// TwinCAT 3 PLC project Untitled1
// ProgramVersion: 3.1.4026.17
// libraries:
//   Tc2_Standard, * (Beckhoff Automation GmbH)
//   Tc2_System, * (Beckhoff Automation GmbH)
// project tree:
//   DUTs/ E_CompressionStages.TcDUT, E_InletToSystem.TcDUT, E_OutletNumber.TcDUT, E_TankBundleNumber.TcDUT, E_ErrorState.TcDUT, E_SolenoidState.TcDUT, ST_AnalogPressureTemp.TcDUT, ST_Path.TcDUT, ST_SolenoidConfig.TcDUT
//   GVLs/ GVL_HMI.TcGVL, GVL_IO.TcGVL
//   / PlcTask.TcTTO
//   POUs/ FB_Device.TcPOU, FB_Matrix.TcPOU, FB_PressureTransducer.TcPOU, FB_Solenoid.TcPOU, MAIN.TcPOU
// real-time tasks:
//   TASK PlcTask: cycle T#10ms, priority 20, ADS port 350
// I/O:
//   DEVICE Node 05 (disabled), AmsNetId 192.168.1.166.2.1
//     Node 05S0 [EK1100 EtherCAT Coupler (2A E-Bus)]
//       Node 05S2 [EL3058 8Ch. Ana. Input 4-20mA]
//       Node 05S4 [EL3058 8Ch. Ana. Input 4-20mA]
//       Node 05S6 [EL3058 8Ch. Ana. Input 4-20mA]
//       Node 05S8 [EL3058 8Ch. Ana. Input 4-20mA]
//       Node 05S10 [EL3058 8Ch. Ana. Input 4-20mA]
//       Node 05S11 [EL1904, 4 Ch. Safety Input 24V, TwinSAFE]
//         modules: Module 1 (FSOES)
//   DEVICE Node 06 (disabled), AmsNetId 192.168.1.166.3.1
//     Node 06S0 [EK1100 EtherCAT Coupler (2A E-Bus)]
//       Node 06S2 [EL2024 4Ch. Dig. Output 24V, 2A]
//       Node 06S4 [EL2024 4Ch. Dig. Output 24V, 2A]
//       Node 06S6 [EL2024 4Ch. Dig. Output 24V, 2A]
//       Node 06S8 [EL2024 4Ch. Dig. Output 24V, 2A]
//       Node 06S10 [EL2024 4Ch. Dig. Output 24V, 2A]
//       Node 06S12 [EL2024 4Ch. Dig. Output 24V, 2A]
//       Node 06S14 [EL2024 4Ch. Dig. Output 24V, 2A]
//       Node 06S16 [EL2024 4Ch. Dig. Output 24V, 2A]
// variable links:
//   Untitled1/Untitled1 Instance <-> Node 05/Node 05S0/Node 05S2
//     PlcTask Inputs/GVL_IO.aPressRaw[{1..8}] <-> AI Standard Channel {1..8}/Value  (8 links)
//   Untitled1/Untitled1 Instance <-> Node 05/Node 05S0/Node 05S4
//     PlcTask Inputs/GVL_IO.aPressRaw[10] <-> AI Standard Channel 2/Value
//     PlcTask Inputs/GVL_IO.aPressRaw[11] <-> AI Standard Channel 3/Value
//     PlcTask Inputs/GVL_IO.aPressRaw[12] <-> AI Standard Channel 4/Value
//     PlcTask Inputs/GVL_IO.aPressRaw[13] <-> AI Standard Channel 5/Value
//     PlcTask Inputs/GVL_IO.aPressRaw[14] <-> AI Standard Channel 8/Value
//     PlcTask Inputs/GVL_IO.aPressRaw[15] <-> AI Standard Channel 6/Value
//     PlcTask Inputs/GVL_IO.aPressRaw[16] <-> AI Standard Channel 7/Value
//     PlcTask Inputs/GVL_IO.aPressRaw[9] <-> AI Standard Channel 1/Value
//   Untitled1/Untitled1 Instance <-> Node 05/Node 05S0/Node 05S6
//     PlcTask Inputs/GVL_IO.aTempRaw[{1..8}] <-> AI Standard Channel {1..8}/Value  (8 links)
//   Untitled1/Untitled1 Instance <-> Node 05/Node 05S0/Node 05S8
//     PlcTask Inputs/GVL_IO.aTempRaw[10] <-> AI Standard Channel 2/Value
//     PlcTask Inputs/GVL_IO.aTempRaw[11] <-> AI Standard Channel 3/Value
//     PlcTask Inputs/GVL_IO.aTempRaw[12] <-> AI Standard Channel 4/Value
//     PlcTask Inputs/GVL_IO.aTempRaw[13] <-> AI Standard Channel 5/Value
//     PlcTask Inputs/GVL_IO.aTempRaw[14] <-> AI Standard Channel 8/Value
//     PlcTask Inputs/GVL_IO.aTempRaw[15] <-> AI Standard Channel 6/Value
//     PlcTask Inputs/GVL_IO.aTempRaw[16] <-> AI Standard Channel 7/Value
//     PlcTask Inputs/GVL_IO.aTempRaw[9] <-> AI Standard Channel 1/Value

CONFIGURATION Untitled1
    RESOURCE PLC ON TwinCAT3
        TASK PlcTask(INTERVAL := T#10ms, PRIORITY := 20);
        PROGRAM MAIN WITH PlcTask : MAIN;
    END_RESOURCE
END_CONFIGURATION

// ---- DUTs/E_CompressionStages.TcDUT
{attribute 'strict'}
TYPE E_CompressionStages :
(
	Bypass_Line:=1,
    Second_Stage_Compression:=2,
    First_Stage_Compression:=3
)USINT;
END_TYPE

// ---- DUTs/E_InletToSystem.TcDUT
{attribute 'qualified_only'}
{attribute 'strict'}
{attribute 'to_string'}
//Pathing Enum
TYPE E_InletToSystem :
(
	Recirculation_From_Storage:=1,Hydrogen_Inlet:=2
);
END_TYPE

// ---- DUTs/E_OutletNumber.TcDUT
{attribute 'strict'}
//Pathing Enum
TYPE E_OutletNumber :
(
	Outlet_2:=1,
    Outlet_1:= 2,
    Recirculation:=3
)USINT;
END_TYPE

// ---- DUTs/E_TankBundleNumber.TcDUT
{attribute 'qualified_only'}
{attribute 'strict'}
{attribute 'to_string'}
//Pathing Enum
TYPE E_TankBundleNumber :
(
	Bundle_Tank_1:=1,Bundle_Tank_2:=2,Bundle_Tank_3:=3,Bundle_Tank_4:=4
);
END_TYPE

// ---- DUTs/E_ErrorState.TcDUT
{attribute 'qualified_only'}
{attribute 'strict'}
{attribute 'to_string'}
TYPE E_ErrorState :
(
	Healthy := 0, Warning:=1, Alarm:= 2, Disabled:=3
);
END_TYPE

// ---- DUTs/E_SolenoidState.TcDUT
{attribute 'qualified_only'}
{attribute 'strict'}
{attribute 'to_string'}
TYPE E_SolenoidState :
(
	Open:=0, Closed:=1
);
END_TYPE

// ---- DUTs/ST_AnalogPressureTemp.TcDUT
TYPE ST_AnalogPressureTemp :
	//Config struct for pressure/temp sensors
STRUCT
	rWarninglevel: REAL;
	rErrorLevel: REAL;
	rPressureMaxSP:REAL;
	rPressureMinSP:REAL;
	rTemperatureMaxSP:REAL;
	rTemperatureMinSP:REAL;
	nRawMax:INT;
	nRawMin:INT;
END_STRUCT
END_TYPE

// ---- DUTs/ST_Path.TcDUT
TYPE ST_Path :
	//Path integer values
STRUCT
	startPath : INT;
	endPath : INT;
END_STRUCT
END_TYPE

// ---- DUTs/ST_SolenoidConfig.TcDUT
TYPE ST_SolenoidConfig :
STRUCT
	NormallyOpen:BOOL; //True if valve to be configured as Normally open
    bOpen:BOOL; //True if valve should be opened
	
END_STRUCT
END_TYPE

// ---- GVLs/GVL_HMI.TcGVL
{attribute 'qualified_only'}
VAR_GLOBAL
	//Variables for the dispensing matrix
	aDispManualValveSelection : ARRAY [1..4,1..3] OF BOOL;
	bDispTurnOnMatrix: BOOL;
	bDispResetMatrix:BOOL;
	bDispTurnOnPathing:BOOL;
	bDispActuatePath:BOOL;
	eDispStartOfPath: E_TankBundleNumber;
	eDispEndOfPath:E_OutletNumber;
	aDispStateofValves: ARRAY[1..cMaxRows,1..cMaxCols] OF E_SolenoidState;
	
	//Variables for the inlet matrix
    aInletManualValveSelection : ARRAY [1..2,1..3] OF BOOL;
	bInletTurnOnMatrix: BOOL;
	bInletResetMatrix:BOOL;
	bInbletTurnOnPathing:BOOL;
	bInletActuatePath:BOOL;
	eInletStartOfPath: E_InletToSystem;
	eInletEndOfPath:E_CompressionStages;
	aInletStateofValves: ARRAY[1..cMaxRows,1..cMaxCols] OF E_SolenoidState;
	
	//Variables for the Filling Matrix
	aFillManualValveSelection : ARRAY [1..4,1..3] OF BOOL;
	bFillTurnOnMatrix: BOOL;
	bFillResetMatrix:BOOL;
	bFillTurnOnPathing:BOOL;
	bFillActuatePath:BOOL;
	eFillStartOfPath: E_TankBundleNumber;
	eFillEndOfPath:E_CompressionStages;
	aFillStateofValves: ARRAY[1..cMaxRows,1..cMaxCols] OF E_SolenoidState;
	
	//Variables to enable and reset Sensors
	bEnableSensors:BOOL;
	bResetSensors:BOOL;
	
	//Sensor Error states
	aSensorErrors :  ARRAY[1..GVL_IO.cNumofPT] OF E_ErrorState;
	
	//Sensor Engineering values
	aPV:  ARRAY[1..GVL_IO.cNumofPT] OF REAL;
	aTV:  ARRAY[1..GVL_IO.cNumofPT] OF REAL;
	
END_VAR
VAR_GLOBAL CONSTANT
	//Set max matrix size at compile time
	cMaxRows:INT:=4;
	cMaxCols:INT:=3;
END_VAR

// ---- GVLs/GVL_IO.TcGVL
{attribute 'qualified_only'}
VAR_GLOBAL CONSTANT
	cNumofPT:USINT:=16;
sPTTags : ARRAY[1..cNumofPT] OF T_MaxString := [
        'PT-301-A-II',
        'PT-302-A-II',
        'PT-350-A-II',
        'PT-351-A-II',
        'PT-352-A-II',
        'PT-353-A-II',
        'PT-354-A-II',
        'PT-355-A-II',
        'PT-356-A-II',
        'PT-357-A-II',
        'PT-358-A-II',
        'PT-359-A-II',
        'PT-360-A-II',
        'PT-365-A-II',
        'PT-361-A-II',
        'PT-363-A-II'
    ];
END_VAR
VAR_GLOBAL
	//Sensor Inputs
	aPressRaw AT %I*: ARRAY[1..cNumofPT] OF INT;
    aTempRaw AT %I* : ARRAY[1..cNumofPT]  OF INT;
	
	//Solenoid Outputs
	aInletMAtrixValveCmds: ARRAY [1..2,1..3] OF BOOL;
	aFillMatrixValveCmds: ARRAY [1..4,1..3] OF BOOL;
	aDispenseMatrixValveCmds: ARRAY [1..4,1..3] OF BOOL;

END_VAR

// ---- POUs/MAIN.TcPOU
PROGRAM MAIN
VAR CONSTANT
	//Constants to set maximum matrix size at compile time
	cMaxRows:INT:=4;
	cMaxCols:INT:=3;
END_VAR
VAR
	//Configure Dispense Matrix [4,3]
	fbDispenseMatrix:FB_Matrix;
	aDispenseMatrixConfig : ARRAY [1..cMaxRows,1..cMaxCols] OF ST_SolenoidConfig;
	bDispMatrixEnable:BOOL;
	bDispMatrixReset:BOOL;
	Disp_st_path : ST_Path;
	bDispFindPath: BOOL;
	bDispPathingSwitch:BOOL;
	nDispenseRows:INT:=4;
	nDispenseCols:INT:=3;
	
	//Configure Inlet Matrix [2,3]
	fbInletMatrix:FB_Matrix;
	aInletMatrixConfig: ARRAY [1..cMaxRows,1..cMaxCols] OF ST_SolenoidConfig;
	bInletMatrixEnable:BOOL;
	bInletMatrixReset:BOOL;
	Inlet_st_path : ST_Path;
	bInletFindPath: BOOL;
	bInletPathingSwitch:BOOL;
	nInletRows:INT:=2;
	nInletCols:INT:=3;
	
	//Configure Filling Matrix [4,3]
	fbFillMatrix:FB_Matrix;
	aFillMatrixConfig : ARRAY [1..cMaxRows,1..cMaxCols] OF ST_SolenoidConfig;
	bFillMatrixEnable:BOOL;
	bFillMatrixReset:BOOL;
	Fill_st_path : ST_Path;
	bFillFindPath: BOOL;
	bFillPathingSwitch:BOOL;
	nFillRows:INT:=4;
	nFillCols:INT:=3;	
	
	//Array of Pressure Transducers
	aPT: ARRAY [1.. GVL_IO.cNumofPT] OF FB_PressureTransducer;
	
	//Standard Config Parameter Struct for Pressure and Temp sensors
	stAnalogCfg : ST_AnalogPressureTemp;
	
	//Initialising Boolean 
	bInitialise:BOOL:=TRUE;
END_VAR

//Run Initialise Method once on first cycle
IF bInitialise THEN
	M_Initalize();
	bInitialise:=FALSE;
END_IF

//Update sensors from IO
M_Sensors();

//Calling FB_MAtrix for each of the three matrices of valves, Dispense, Inlet and FIlling.
fbDispenseMatrix(bDeviceEnable:=bDispMatrixEnable,bDeviceReset:=bDispMatrixReset,
	            aConfig:=aDispenseMatrixConfig,st_path:=Disp_st_path,bSetCurrentPath:=bDispFindPath,
                bPathingOn:=bDispPathingSwitch,nRowSize:=nDispenseRows,nColSize:=nDispenseCols);
				
fbInletMatrix(bDeviceEnable:=bInletMatrixEnable,bDeviceReset:=bInletMatrixReset,aConfig:=aInletMatrixConfig,
	          st_path:=Inlet_st_path,bSetCurrentPath:=bInletFindPath,bPathingOn:=bInletPathingSwitch,
			  nRowSize:=nInletRows,nColSize:=nInletCols);
			  
fbFillMatrix(bDeviceEnable:=bFillMatrixEnable,bDeviceReset:=bFillMatrixReset,aConfig:=aFillMatrixConfig,
	          st_path:=Fill_st_path,bSetCurrentPath:=bFillFindPath,bPathingOn:=bFillPathingSwitch,
			  nRowSize:=nFillRows,nColSize:=nFillCols);

				
//Update the inputs to the matrix functions and pressure sensors from GVLs
M_UpdateFromHMI();

METHOD M_ActuateValves
VAR_INPUT
	rows:INT;
	cols:INT;
END_VAR
END_METHOD

METHOD PUBLIC M_Initalize 
VAR
rows:INT;
cols:INT;
END_VAR

//Configure the pressure sensors
	stAnalogCfg.rWarninglevel:=500;
	stAnalogCfg.rErrorLevel:=525;
	stAnalogCfg.rPressureMinSP:=0;
	stAnalogCfg.rPressureMaxSP:=1000;
	stAnalogCfg.rTemperatureMinSP:=-40;
	stAnalogCfg.rTemperatureMaxSP:=125;
	stAnalogCfg.nRawMin:=0;
	stAnalogCfg.nRawMax:=32767;
//Configure the pressure sensors
FOR rows:=1 TO GVL_IO.cNumofPT DO
    aPT[rows].st_AnalogPressureTempdata:=stAnalogCfg;
	apT[rows].sTag:=GVL_IO.sPTTags[rows];
END_FOR


//Initialise all matrices to be NC and to be un-energised
    FOR  rows:=1 TO cMaxRows DO
       FOR  cols:=1 TO cMaxCols DO
          aDispenseMatrixConfig[rows,cols].NormallyOpen:=FALSE;
		  aInletMatrixConfig[rows,cols].NormallyOpen:=FALSE;
		  aDispenseMatrixConfig[rows,cols].bOpen:=FALSE;
		  aInletMatrixConfig[rows,cols].bOpen:=FALSE;
		  aFillMatrixConfig[rows,cols].NormallyOpen:=FALSE;
		  aFillMatrixConfig[rows,cols].bOpen:=FALSE;
       END_FOR
    END_FOR
END_METHOD

METHOD M_Sensors
VAR
	nsensorNumber:INT;
END_VAR
FOR nsensorNumber:=1 TO GVL_IO.cNumofPT DO
	aPT[nsensorNumber](bDeviceEnable:=GVL_HMI.bEnableSensors,
		               bDeviceReset:=GVL_HMI.bResetSensors,
					   nSensorPressure:=GVL_IO.aPressRaw[nsensorNumber],
					   nSensorTemperature:=GVL_IO.aTempRaw[nsensorNumber],
					   rEngPressure=>GVL_HMI.aPV[nsensorNumber],
					   rEngTemperature=>GVL_HMI.aTV[nsensorNumber],
                       eDeviceState=>GVL_HMI.aSensorErrors[nsensorNumber]);			   
END_FOR
END_METHOD

METHOD M_UpdateDispenseFromHMI
VAR
	rows:INT;
	cols:INT;
END_VAR
//Variables for actuating the Dispense matrix updated from GVL here
bDispMatrixEnable:=GVL_HMI.bDispTurnOnMatrix;
bDispMatrixReset:=GVL_HMI.bDispResetMatrix;
Disp_st_path.endPath:=GVL_HMI.eDispEndOfPath;
Disp_st_path.startPath:=GVL_HMI.eDispStartOfPath;
bDispFindPath:=GVL_HMI.bDispActuatePath;
bDispPathingSwitch:=GVL_HMI.bDispTurnOnPathing;

//Change the display state of the matrix valves on the HMI screen
GVL_HMI.aDispStateofValves:=fbDispenseMatrix.aValveStates;

//Condition to avoid manual control when pathing is on
IF GVL_HMI.bDispTurnOnPathing THEN
	RETURN;
END_IF
FOR rows := 1 TO nDispenseRows DO
       FOR cols := 1 TO nDispenseCols DO
          aDispenseMatrixConfig[rows,cols].bOpen:=GVL_HMI.aDispManualValveSelection[rows,cols];
       END_FOR
END_FOR
END_METHOD

METHOD M_UpdateFillFromHMI
VAR
	rows:INT;
	cols:INT;
END_VAR
//Variables for actuating the filling matrix are updated from GVL here
bFillMatrixEnable:=GVL_HMI.bFillTurnOnMatrix;
bFillMatrixReset:=GVL_HMI.bFillResetMatrix;
bFillFindPath:=GVL_HMI.bFillActuatePath;
bFillPathingSwitch:=GVL_HMI.bFillTurnOnPathing;
Fill_st_path.endPath:=GVL_HMI.eFillEndOfPath;
Fill_st_path.startPath:=GVL_HMI.eFillStartOfPath;

//Change the display state of the matrix valves on the HMI screen
GVL_HMI.aFillStateofValves:=fbFillMatrix.aValveStates;


//Condition to avoid manual control when pathing is on
IF GVL_HMI.bFillTurnOnPathing THEN
	RETURN;
END_IF
FOR rows := 1 TO nFillRows DO
       FOR cols := 1 TO nFillCols DO
          aFillMatrixConfig[rows,cols].bOpen:=GVL_HMI.aFillManualValveSelection[rows,cols];
       END_FOR
END_FOR
END_METHOD

METHOD M_UpdateFromHMI
//Update each matrix Independently
M_UpdateDispenseFromHMI();
M_UpdateInletFromHMI();
M_UpdateFillFromHMI();
END_METHOD

METHOD M_UpdateInletFromHMI
VAR
	rows:INT;
	cols:INT;
END_VAR
//Variables for actuating the inlet matrix are updated from the GVL here
bInletMatrixEnable:=GVL_HMI.bInletTurnOnMatrix;
bInletMatrixReset:=GVL_HMI.bInletResetMatrix;
bInletFindPath:=GVL_HMI.bInletActuatePath;
bInletPathingSwitch:=GVL_HMI.bInbletTurnOnPathing;
Inlet_st_path.endPath:=GVL_HMI.eInletEndOfPath;
Inlet_st_path.startPath:=GVL_HMI.eInletStartOfPath;

//Change the display state of the matrix valves on the HMI screen
GVL_HMI.aInletStateofValves:=fbInletMatrix.aValveStates;

//Condition to avoid manual control when pathing is on
IF GVL_HMI.bInbletTurnOnPathing THEN
	RETURN;
END_IF
FOR rows := 1 TO nInletRows DO
       FOR cols := 1 TO nInletCols DO
          aInletMatrixConfig[rows,cols].bOpen:=GVL_HMI.aInletManualValveSelection[rows,cols];
       END_FOR
END_FOR
END_METHOD

END_PROGRAM

// ---- POUs/FB_Matrix.TcPOU
FUNCTION_BLOCK FB_Matrix EXTENDS FB_Device
VAR_INPUT
	st_path : ST_Path;//INT struct to contain int value of path enums
	bSetCurrentPath:BOOL;//Bool to actuate the selected path 
	bPathingOn:BOOL;//BOOL to enable the path selection mode 
	nRowSize:INT;//Matrix row size 
	nColSize:INT;//Matrix Column size
END_VAR
VAR
	aValves:ARRAY [1..4,1..3] OF FB_Solenoid;//Instantiating Solenoid valves, max array size, can contain smaller arrays
	iRows:INT;//Row variable for FOR loops to use
	iColumns:INT;//Col variable for FOR loops to use
	bOverallEnable:BOOL;//Internal variable used to assign device state to all instantiated solenoid valves
END_VAR
VAR_IN_OUT
	aConfig:ARRAY[1..4,1..3] OF ST_SolenoidConfig;//Matrix config
END_VAR
VAR_OUTPUT
	aValveStates : ARRAY [1..4,1..3] OF E_SolenoidState;//State of valves
	aValveCommands:ARRAY [1..4,1..3] OF BOOL;
END_VAR

M_EnableResetLogic();
M_CyclicLogic();
IF bPathingOn THEN
	M_DispensePathing();
ELSE
	M_ManualControl();
END_IF

METHOD M_CyclicLogic : HRESULT
//Call FB_Device M_Cyclic Logic
hr:=SUPER^.M_CyclicLogic();
 IF bDeviceEnable THEN
   FOR iRows := 1 TO nRowSize DO
       FOR iColumns := 1 TO nColSize DO
           aValves[iRows, iColumns](bDeviceEnable:=bOverallEnable,
		   bNormallyOpen:=aConfig[iRows,iColumns].NormallyOpen,
           bCmdOpen:=aConfig[iRows,iColumns].bOpen,bCoilEnergiseState=>aValveCommands[iRows,iColumns]);
       END_FOR
   END_FOR
   
 ELSE
	 FOR iRows := 1 TO nRowSize DO
       FOR iColumns := 1 TO nColSize DO
           aValves[iRows, iColumns](bDeviceEnable:=bOverallEnable);
       END_FOR
     END_FOR
 END_IF
 
FOR iRows := 1 TO nRowSize DO
   FOR iColumns := 1 TO nColSize DO
       aValveStates[iRows, iColumns]:=aValves[iRows, iColumns].eSolenoidState;
   END_FOR
END_FOR
END_METHOD

METHOD M_DispensePathing : BOOL
VAR
	nRowToOpen: INT :=(st_path.startPath);
	nColToOpen: INT :=(st_path.endPath);
END_VAR
IF bDeviceEnable THEN
	IF bSetCurrentPath THEN
       aConfig[nRowToOpen,nColToOpen].bOpen:=TRUE;
    END_IF
END_IF
END_METHOD

METHOD M_EnableResetLogic : BOOL
//Set up variables and logic to reset and enable valve FB's created by FB_Matrix
bOverallEnable:=bDeviceEnable;
IF bDeviceReset THEN
    FOR iRows := 1 TO nRowSize DO
       FOR iColumns := 1 TO nColSize DO
           aValves[iRows, iColumns](bDeviceReset:=fbTrig.Q);
		   aConfig[iRows,iColumns].bOpen:=FALSE;
		   GVL_HMI.aDispManualValveSelection[iRows,iColumns]:=FALSE;
		   GVL_HMI.aInletManualValveSelection[iRows,iColumns]:=FALSE;
		   GVL_HMI.aFillManualValveSelection[iRows,iColumns]:=FALSE;
       END_FOR
    END_FOR
END_IF
END_METHOD

METHOD M_ManualControl
IF NOT bPathingOn AND bDeviceEnable THEN
   FOR iRows := 1 TO 4 DO
       FOR iColumns := 1 TO 3 DO
           aValves[iRows, iColumns](bCmdOpen:=aConfig[iRows,iColumns].bOpen);
       END_FOR
   END_FOR
END_IF
END_METHOD

END_FUNCTION_BLOCK

// ---- POUs/FB_Device.TcPOU
FUNCTION_BLOCK PUBLIC FB_Device
VAR_INPUT
	bDeviceEnable:BOOL; //Make the device Active
	bDeviceReset:BOOL;//Reset Error state
END_VAR
VAR_OUTPUT
    bError        : BOOL;   // True if in error
	bWarning :BOOL; //True if warning applicable
    eDeviceState  : E_ErrorState; // Summary device state
END_VAR
VAR
	hr : HRESULT;
	fbTrig:R_TRIG;
END_VAR

hr := M_CyclicLogic();

METHOD PUBLIC M_CyclicLogic : HRESULT
//  Check enable state
IF NOT bDeviceEnable THEN
	eDeviceState:=E_ErrorState.Disabled;
	M_CyclicLogic := S_Pending;
	RETURN;
END_IF

// Check reset 
fbTrig(CLK:=bDeviceReset);
IF fbTrig.Q THEN
	bError:=FALSE;
	bWarning:=FALSE;
	eDeviceState:=E_ErrorState.Healthy;
END_IF

// Handle state logic
IF bError THEN
	eDeviceState:=E_ErrorState.Alarm;
ELSIF bWarning THEN
        eDeviceState:=E_ErrorState.Warning;	
ELSE 
		eDeviceState:=E_ErrorState.Healthy;
END_IF

M_CyclicLogic := S_OK;
END_METHOD

END_FUNCTION_BLOCK

// ---- POUs/FB_Solenoid.TcPOU
FUNCTION_BLOCK FB_Solenoid EXTENDS FB_Device
VAR_INPUT
	bNormallyOpen:BOOL;//True if Valve is Normally Open
	bCmdOpen:BOOL;// True if Valve should be opened
END_VAR
VAR
	bTheoreticallyOpen:BOOL;
END_VAR
VAR_OUTPUT
	bCoilEnergiseState:BOOL;//Signal sent to coil to energise
	eSolenoidState: E_SolenoidState;//If coil is not energised in reality
END_VAR

IF bCmdOpen THEN
	M_Open();
ELSE
    M_Close();
END_IF

METHOD M_CheckState
IF bTheoreticallyOpen THEN
	eSolenoidState := E_SolenoidState.Open;
ELSE
	eSolenoidState := E_SolenoidState.Closed;
END_IF
END_METHOD

METHOD PUBLIC M_Close : HRESULT
hr:=SUPER^.M_CyclicLogic();
IF bDeviceEnable THEN
	IF bNormallyOpen THEN
		bCoilEnergiseState := TRUE;
		bTheoreticallyOpen := FALSE;
	ELSE
		bCoilEnergiseState := FALSE;
		bTheoreticallyOpen := bNormallyOpen;
	END_IF
ELSE
	bCoilEnergiseState := FALSE;
	bTheoreticallyOpen := bNormallyOpen;
END_IF
M_CheckState();
END_METHOD

METHOD PUBLIC M_Open : HRESULT
hr:=SUPER^.M_CyclicLogic();
IF bDeviceEnable THEN
	IF NOT bNormallyOpen THEN
		bCoilEnergiseState := TRUE;
		bTheoreticallyOpen := TRUE;
	ELSE
		bCoilEnergiseState := FALSE;
		bTheoreticallyOpen := bNormallyOpen;
	END_IF
ELSE
	bCoilEnergiseState := FALSE;
	bTheoreticallyOpen := bNormallyOpen;
END_IF
M_Checkstate();
END_METHOD

END_FUNCTION_BLOCK

// ---- POUs/FB_PressureTransducer.TcPOU
FUNCTION_BLOCK FB_PressureTransducer EXTENDS FB_Device
VAR_INPUT
	nSensorPressure: INT; //Pressure analog input
	nSensorTemperature:INT;//Temperature analog input 
	st_AnalogPressureTempdata:ST_AnalogPressureTemp;//Configuration struct 
	sTag : T_MaxString;
END_VAR
VAR_OUTPUT
	rEngPressure:REAL;//Pressure in BAR.
	rEngTemperature:REAL;//Temperature in Degrees C.
END_VAR

M_CyclicLogic();

METHOD M_CyclicLogic : HRESULT
VAR
	rNormPressure:REAL;
	rNormTemperature:REAL;
END_VAR
//Call M_CyclicLogic from FB_Device 
hr:=SUPER^.M_CyclicLogic();
IF bDeviceEnable THEN
	//Normalise the analog inputs 
   rNormPressure    := (INT_TO_REAL(nSensorPressure)    - INT_TO_REAL(st_AnalogPressureTempdata.nRawMin)) / (INT_TO_REAL(st_AnalogPressureTempdata.nRawMax) - INT_TO_REAL(st_AnalogPressureTempdata.nRawMin));
   rNormTemperature := (INT_TO_REAL(nSensorTemperature) - INT_TO_REAL(st_AnalogPressureTempdata.nRawMin)) / (INT_TO_REAL(st_AnalogPressureTempdata.nRawMax) - INT_TO_REAL(st_AnalogPressureTempdata.nRawMin));
   
   //Scale analog inputs to the Engineering process values, using config struct parameters
   rEngPressure:=st_AnalogPressureTempdata.rPressureMinSP + rNormPressure * (st_AnalogPressureTempdata.rPressureMaxSP - st_AnalogPressureTempdata.rPressureMinSP);
   rEngTemperature:=st_AnalogPressureTempdata.rTemperatureMinSP + rNormTemperature * (st_AnalogPressureTempdata.rTemperatureMaxSP - st_AnalogPressureTempdata.rTemperatureMinSP);
END_IF

//Evaluate pressure state 
M_PressureState();
END_METHOD

METHOD M_PressureState : BOOL
//Evaluate pressure value against warning and error values.
IF (rEngPressure > 500) AND (rEngPressure < 525) THEN
	bWarning:=TRUE;
ELSIF rEngPressure > 525 THEN
	bError:=TRUE;
ELSE 
	bWarning:=FALSE;
END_IF
END_METHOD

END_FUNCTION_BLOCK
